TYPE T_FOD_Cur :
STRUCT
END_STRUCT
END_TYPE

(* stored: Version 1.1.0.1, ProductVersion 3.1.0.23
   DUT T_FOD_Cur: Id {644c02d4-3e0c-4b06-a136-9b70a31efa14} *)
